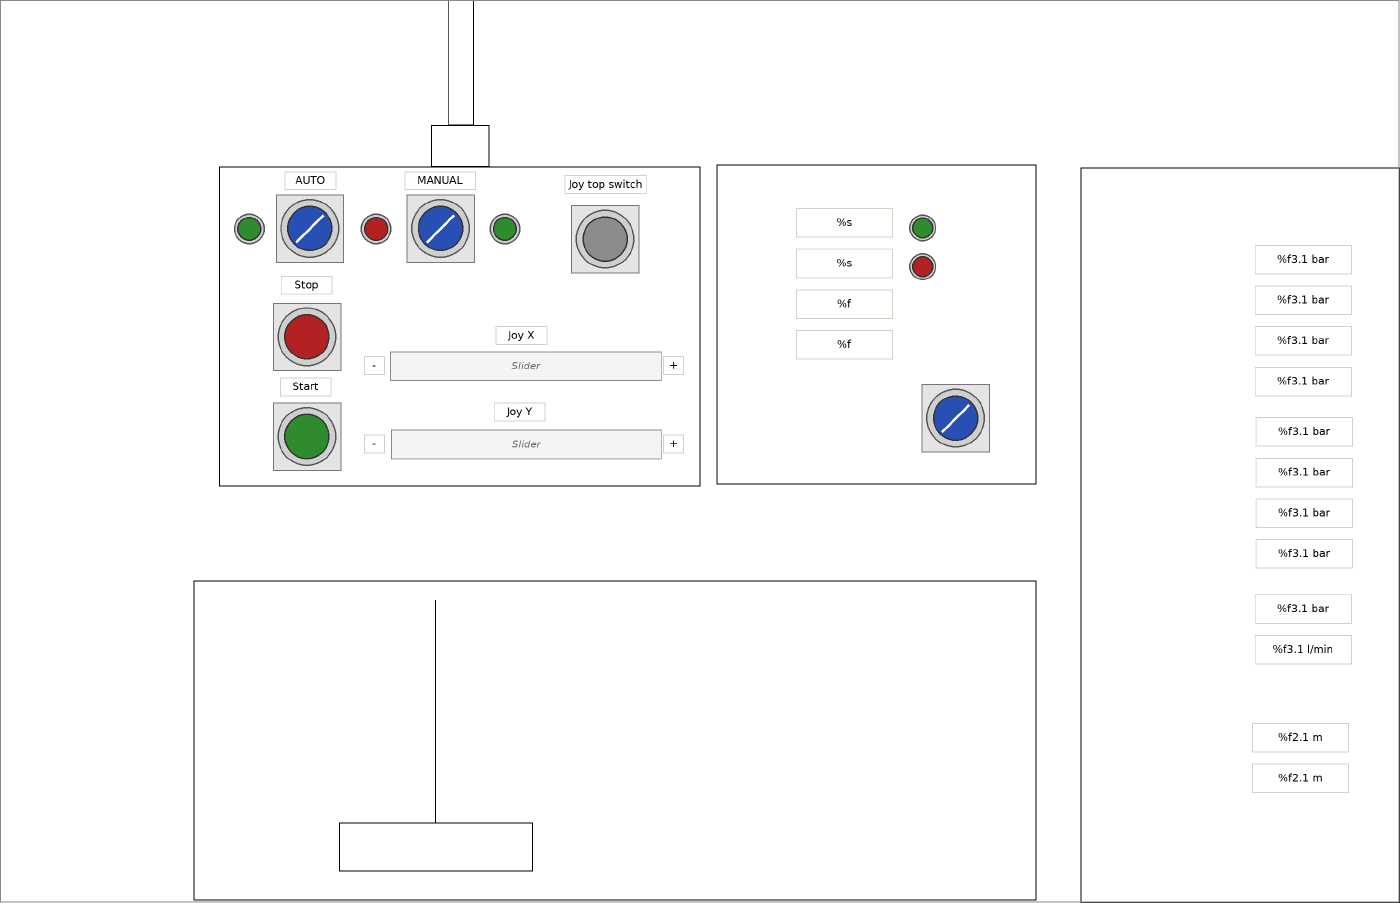
VISUALIZATION Visualization  // 1446x933
    RoundedRectangle (226,172 497x330)
    RotarySwitch (285,201 70x70), variable: G_ControlBox.bAuto, behaviour: TOGGLE, style: Switch-RotarySwitch-Blue
    PushSwitch (282,416 70x70), variable: G_ControlBox.bStart, behaviour: TAP, style: Switch-PushSwitch-Green
    PushSwitch (282,313 70x70), variable: G_ControlBox.bStop, behaviour: TAP, style: Switch-PushSwitch-Red
    RotarySwitch (420,201 70x70), variable: G_ControlBox.bManual, behaviour: TOGGLE, style: Switch-RotarySwitch-Blue
    Slider (404,444 279x30), variable: G_ControlBox.fJoyY, input disabled if: G_ControlBox.bJoyNotActive, scale 0..0
    Slider (403,363 280x30), variable: G_ControlBox.fJoyX, input disabled if: G_ControlBox.bJoyNotActive, scale 0..0
    Rectangle (445,129 60x43)
    Rectangle (463,0 26x129)
    Textfield (290,285 53x19), "Stop"
    Textfield (289,390 53x19), "Start"
    Textfield (512,337 53x19), "Joy X"
    Textfield (510,416 53x19), "Joy Y"
    Textfield (583,181 85x19), "Joy top switch"
    Textfield (685,368 21x19), "+"
    Textfield (685,449 21x19), "+"
    Textfield (376,449 21x19), "-"
    Textfield (376,368 21x19), "-"
    Textfield (294,177 53x19), "AUTO"
    Textfield (418,177 73x19), "MANUAL"
    RoundedRectangle (740,170 330x330)
    Label (756,214 63x30), "Mode:"
    Label (738,253 90x38), "Status:"
    Textfield (822,215 100x30), "%s", text variable: G_ControlBox.eMode
    Lamp1 (937,215 32x41), variable: G_ControlBox.bRunning, style: Lamp-Lamp1-Green
    Textfield (822,257 100x30), "%s", text variable: G_ControlBox.eStatus
    Lamp1 (937,255 32x41), variable: G_ControlBox.bStopping, style: Lamp-Lamp1-Red
    Lamp1 (239,216 37x41), variable: G_ControlBox.bAuto, style: Lamp-Lamp1-Green
    Lamp1 (370,216 37x41), variable: G_ControlBox.bFault, style: Lamp-Lamp1-Red
    Lamp1 (503,216 37x41), variable: G_ControlBox.bManual, style: Lamp-Lamp1-Green
    Textfield (822,299 100x30), "%f", text variable: G_ControlBox.fJoyX_Normalized
    Textfield (822,341 100x30), "%f", text variable: G_ControlBox.fJoyY_Normalized
    Label (780,298 45x38), "X:"
    Label (780,337 45x38), "Y:"
    RoundedRectangle (200,600 870x330)
    Rectangle (350,850 200x50)
        p3528305787: G_Sim.nX
        p2773130477: G_Sim.nY
        p874137650: G_Sim.nX
        p1126004900: G_Sim.nY
    Line (450,850) (450,620)
        p3528305787: G_Sim.nX
        p874137650: G_Sim.nX
        p2773130477: G_Sim.nY
    PushSwitchLed (590,212 70x70), variable: G_ControlBox.bJoyActive, behaviour: TOGGLE, style: Switch-PushSwitchLed-Gray
    RoundedRectangle (1116,173 330x760)
    Label (1205,252 88x30), "Supply"
    Label (1200,291 102x38), "Return"
    Textfield (1296,253 100x30), "%f3.1 bar", text variable: G_HMI.n_pS
    Textfield (1296,295 100x30), "%f3.1 bar", text variable: G_HMI.n_pR
    Textfield (1296,337 100x30), "%f3.1 bar", text variable: G_HMI.n_pCA
    Textfield (1296,379 100x30), "%f3.1 bar", text variable: G_HMI.n_pCB
    Label (1156,336 143x38), "Cylinder rod"
    Label (1137,375 162x38), "Cylinder piston"
    Label (1193,430 101x30), "Winch in"
    Label (1123,469 180x38), "Winch in before"
    Textfield (1297,431 100x30), "%f3.1 bar", text variable: G_HMI.n_pWA
    Textfield (1297,473 100x30), "%f3.1 bar", text variable: G_HMI.n_pWA1
    Textfield (1297,515 100x30), "%f3.1 bar", text variable: G_HMI.n_pWA1
    Textfield (1297,557 100x30), "%f3.1 bar", text variable: G_HMI.n_pWB
    Label (1176,514 124x38), "Winch out"
    Label (1141,553 159x38), "Winch out red"
    Label (1164,613 129x30), "Winch drain"
    Label (1163,652 139x38), "Winch flow"
    Textfield (1296,614 100x30), "%f3.1 bar", text variable: G_HMI.n_pWD
    Textfield (1296,656 100x30), "%f3.1 l/min", text variable: G_HMI.n_QW
    Textfield (1293,747 100x30), "%f2.1 m", text variable: G_HMI.n_Xc
    Textfield (1293,789 100x30), "%f2.1 m", text variable: G_HMI.n_WinchEncoder
    Label (1156,746 140x38), "Cylinder pos"
    Label (1160,785 136x38), "Load height"
    RotarySwitch (952,397 70x70), variable: G_ControlBox.bAuto, behaviour: TOGGLE, style: Switch-RotarySwitch-Blue
    Label (1145,198 194x38), "Pressures:"
    Label (1125,700 251x38), "Position:"
END_VISUALIZATION

(* stored: Version 1.1.0.1, ProductVersion 3.1.4024.12
   Visu Visualization: Id {81918428-894a-4d31-8869-aaee674000f5} *)
